// TIA Portal project "RollDice" (V17)

(* hardware
DEVICE "HMI_1"  TP1500 Comfort
   slot 0: "HMI_1"  TP1500 Comfort  6AV2 124-0QC02-0AX0  17.0.0.0
   slot 1: "HMI_RT_1"  TP1500 Comfort  6AV2 124-0QC02-0AX0  17.0.0.0
   slot 5: "HMI_1.IE_CP_1"  PROFINET Interface  17.0.0.0
      slot 1: "PROFINET Interface_1"  PROFINET Interface
         slot 1: "Port_1"  Port
         slot 2: "Port_2"  Port
   slot 6: "HMI_1.IE_CP_2"  PROFINET Interface  17.0.0.0
      slot 1: "PROFINET Interface_GBit"  PROFINET Interface
         slot 1: "Port_1"  Port
   slot 7: "HMI_1.MPI/DP_CP_1"  MPI/DP Interface  17.0.0.0
DEVICE "S7-1500/ET200MP station_1"  S7-1500 station
   slot 0: "Rail_0"  Rack  6ES7 590-1***0-0AA0
   slot 1: "PLC_1"  CPU 1515-2 PN  6ES7 515-2AM02-0AB0  V2.9
      slot 3: "CPU display_1"  6ES7591-1BA00-0AA0
      slot 32768: "PROFINET interface_1"  X1
         slot 32769: "Port_1"  X1 P1
         slot 32770: "Port_2"  X1 P2
      slot 33024: "PROFINET interface_2"  X2
         slot 33025: "Port_1"  X2 P1
      slot 34817: "Virtual CP interface port_1"  Virtual CP interface port  Virtual CP interface port
*)

// ===== PLC "PLC_1"  CPU 1515-2 PN =====

TYPE "Dice_PLCD"
   STRUCT
      Number : Int;   // 1-6 => Number on the Dice
      xRolled : Bool;   // True=> Dice has been clicked
   END_STRUCT;
END_TYPE

DATA_BLOCK "MainDB"   // DB1
{ S7_Optimized_Access := 'TRUE' }
VERSION : 0.1
   VAR
      Dice : Array[0..6] of "Dice_PLCD";
   END_VAR
BEGIN
END_DATA_BLOCK

FUNCTION "Dice_FC" : Void   // FC1, SCL
{ S7_Optimized_Access := 'TRUE' }
VERSION : 0.1
   VAR_OUTPUT
      error : Bool;   // Error if true
      status : Word;   // Status of the function
      subfunctionStatus : Word;   // Status or return value of called FB's, FCs and system blocks
   END_VAR
   VAR_IN_OUT
      Dice : "Dice_PLCD";
   END_VAR
   VAR_TEMP
      tempTime : DTL;   // System time
      tempNanoSecondInDWord : DWord;   // UDINT converted to DWORD for access to individual bytes
      tempTimeStatus : Word;   // Status of the instruction RD_SYS_T
      tempRandomValue : DWord;   // Random-start-value
      tempNormReal : Real;   // Normalized value
   END_VAR
   VAR CONSTANT
      ZERO : Int := 0;   // Zero value in case of error
      MAX_UDINT : UDInt := 4294967295 ;   // Maximum UDINT value
      SUB_STATUS_NO_ERROR : Word := 16#0000;   // Status: sub function call ends without error
      STATUS_FINISHED_NO_ERROR : Word := 16#0000;   // Status: Execution finished without errors
      ERR_MAX_LESS_MIN : Word := 16#8200;   // Error: The maximum limit number is smaller than the minimum limit number
      ERR_RD_SYS_T : Word := 16#8600;   // Error: System function Read system time returned an error
      LOWEST_NUMBER : UDInt := 1;   // Lowest Number a Dive can Roll
      HIGHEST_NUMBER : UDInt := 6;   // Highest Number a Dive can Roll
   END_VAR
BEGIN
   REGION Block_Header
       // Statement section REGION

   END_REGION

   REGION Validation

       // When not Rolled Jump Out of the Block
       IF #Dice.xRolled <> TRUE THEN
           RETURN;
       END_IF;


       // Read system time
       #tempTimeStatus := INT_TO_WORD(RD_SYS_T(#tempTime));

       // Check return variable for error
       IF (#tempTimeStatus <> #SUB_STATUS_NO_ERROR) THEN
           #error := true;
           #status := #ERR_RD_SYS_T;
           #subfunctionStatus := #tempTimeStatus;
           #Dice.Number := #ZERO;
           RETURN;
       END_IF;
   END_REGION

   REGION Calculating random number
       // Converting to double word so individual bytes can be addressed
       #tempNanoSecondInDWord := UDINT_TO_DWORD(#tempTime.NANOSECOND);

       // Callculate a random-start-value depending on the time
       #tempRandomValue.%B3 := #tempNanoSecondInDWord.%B0;
       #tempRandomValue.%B2 := #tempNanoSecondInDWord.%B1;
       #tempRandomValue.%B1 := #tempNanoSecondInDWord.%B2;
       #tempRandomValue.%B0 := #tempNanoSecondInDWord.%B3;
       // Norm the calculated random number: 0.0 <= #tempNormReal <= 1.0
       #tempNormReal := UDINT_TO_REAL(DWORD_TO_UDINT(#tempRandomValue)) / UDINT_TO_REAL(#MAX_UDINT);

       // Scale the tempNormReal to be in the range of maxValue and minValue
       #Dice.Number := REAL_TO_INT((#tempNormReal * UDINT_TO_REAL(#HIGHEST_NUMBER - #LOWEST_NUMBER) + UDINT_TO_REAL(#LOWEST_NUMBER)));
       #Dice.xRolled := FALSE;
       #error := false;
       #status := #STATUS_FINISHED_NO_ERROR;
       #subfunctionStatus := #SUB_STATUS_NO_ERROR;

       // ENO mechanism is not used
       ENO := TRUE;
   END_REGION
END_FUNCTION

ORGANIZATION_BLOCK "Main"   // OB1, FBD, ProgramCycle
TITLE = "Main Program Sweep (Cycle)"
{ S7_Optimized_Access := 'TRUE' }
VERSION : 0.1
   VAR_INPUT
      Initial_Call : Bool;   // Initial call of this OB
      Remanence : Bool;   // =True, if remanent data are available
   END_VAR
   VAR_TEMP
      Error : Word;
      xError : Bool;
   END_VAR
   VAR_TEMP   // added for the SCL form of the ladder/FBD networks
      _w1 : Bool;
      _w2 : Bool;
      _w3 : Bool;
      _w4 : Bool;
   END_VAR
BEGIN

REGION Network 1: True=> Dice has been clicked
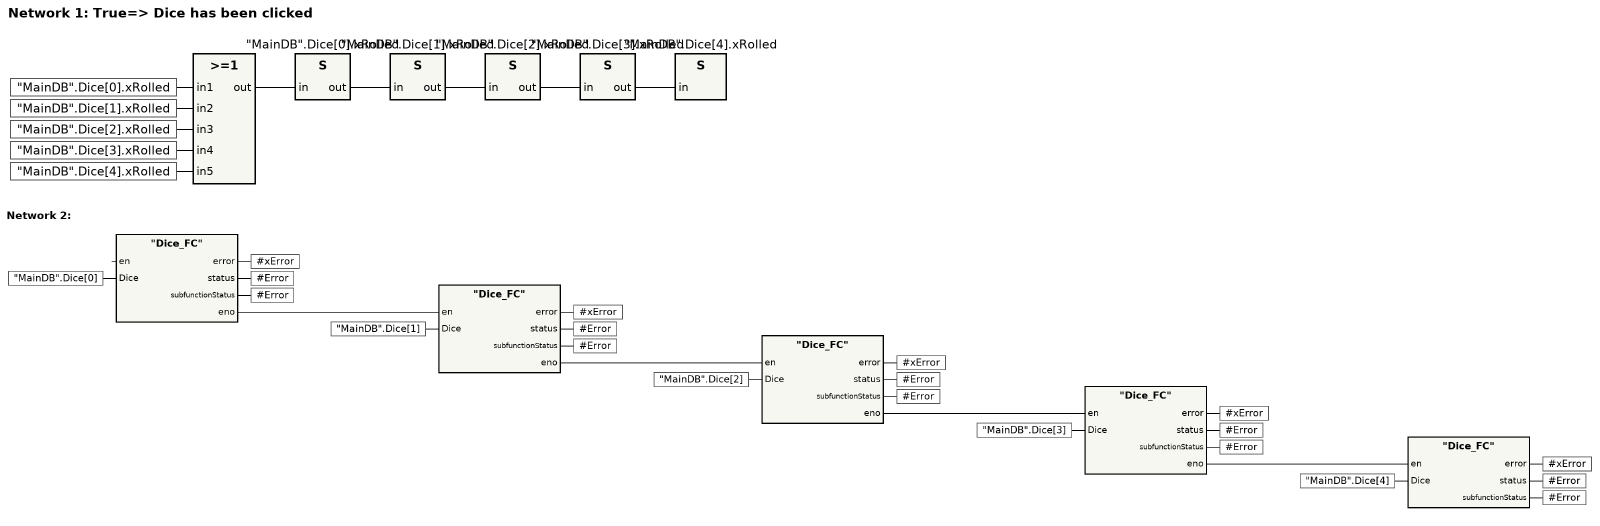
   #_w1 := "MainDB".Dice[0].xRolled OR "MainDB".Dice[1].xRolled OR "MainDB".Dice[2].xRolled OR "MainDB".Dice[3].xRolled OR "MainDB".Dice[4].xRolled;
   IF #_w1 THEN
       "MainDB".Dice[0].xRolled := TRUE;
       "MainDB".Dice[1].xRolled := TRUE;
       "MainDB".Dice[2].xRolled := TRUE;
       "MainDB".Dice[3].xRolled := TRUE;
       "MainDB".Dice[4].xRolled := TRUE;
   END_IF;
END_REGION

REGION Network 2
   "Dice_FC"(Dice := "MainDB".Dice[0],
             error => #xError,
             status => #Error,
             subfunctionStatus => #Error,
             ENO => #_w1);
   "Dice_FC"(EN := #_w1,
             Dice := "MainDB".Dice[1],
             error => #xError,
             status => #Error,
             subfunctionStatus => #Error,
             ENO => #_w2);
   "Dice_FC"(EN := #_w2,
             Dice := "MainDB".Dice[2],
             error => #xError,
             status => #Error,
             subfunctionStatus => #Error,
             ENO => #_w3);
   "Dice_FC"(EN := #_w3,
             Dice := "MainDB".Dice[3],
             error => #xError,
             status => #Error,
             subfunctionStatus => #Error,
             ENO => #_w4);
   IF #_w4 THEN
       "Dice_FC"(Dice := "MainDB".Dice[4], error => #xError, status => #Error, subfunctionStatus => #Error);
   END_IF;
END_REGION
END_ORGANIZATION_BLOCK

// ===== library types =====

// folder: LGF/4 Math operations

FUNCTION "LGF_RandomRange_Dint" : DInt   // FC10013, SCL
TITLE = LGF_RandomRange_DInt
{ S7_Optimized_Access := 'TRUE' }
AUTHOR : Siemens_Digital_Industries
FAMILY : LGF
NAME : LGF_RandomRange_DInt
// This function generates random numbers in defined limits (Datatype DInt)
   VAR_INPUT
      minValue : DInt;   // minimal Value random can reach / Minimum value of the range of the random number
      maxValue : DInt;   // maximal Value random can reach / Maximum value of the range of the random number
   END_VAR
   VAR_OUTPUT
      error : Bool;   // Error if true
      status : Word;   // Status of the function
      subfunctionStatus : Word;   // Status or return value of called FB's, FCs and system blocks
   END_VAR
   VAR_TEMP
      tempTime : DTL;   // System time
      tempNanoSecondInDWord : DWord;   // UDINT converted to DWORD for access to individual bytes
      tempTimeStatus : Word;   // Status of the instruction RD_SYS_T
      tempRandomValue : DWord;   // Random-start-value
      tempNormReal : Real;   // Normalized value
   END_VAR
   // Ret_Val : Returns random DInt number in a predefined range
   VAR CONSTANT
      ZERO : DInt := 0;   // Zero value in case of error
      MAX_UDINT : UDInt := 4294967295 ;   // Maximum UDINT value
      SUB_STATUS_NO_ERROR : Word := 16#0000;   // Status: sub function call ends without error
      STATUS_FINISHED_NO_ERROR : Word := 16#0000;   // Status: Execution finished without errors
      ERR_MAX_LESS_MIN : Word := 16#8200;   // Error: The maximum limit number is smaller than the minimum limit number
      ERR_RD_SYS_T : Word := 16#8600;   // Error: System function Read system time returned an error
   END_VAR
BEGIN
   REGION Block info header
     //=============================================================================
     // SIEMENS AG / (c)Copyright 2017
     //-----------------------------------------------------------------------------
     // Title:            LGF_RandomRange_DInt
     // Comment/Function: This function generates random numbers in defined limits (Datatype DInt)
     // Library/Family:   LGF(Library General Functions)
     // Author:           Siemens Digital Industry Support
     // Tested with:      S7-PLCSIM Advanced V2.0 SP1
     // Engineering:      TIA Portal V15 Update 2
     // Restrictions:     ENO disabled - error handling done by error and status
     // Requirements:     PLC (S7-1200 / S7-1500)
     //-------------------------------------------------------------------------------
     // Change log table:
     // Version  | Date       | Expert in charge       | Changes applied
     //----------|------------|------------------------|------------------------------
     // 01.00.00 19.08.2015  Siemens Industry Online Support
     //                      First released version
     // 01.00.01 02.01.2017  Siemens Industry Online Support
     //                      Upgrade: TIA Portal V14 Update 1
     // 01.00.02 17.08.2018  Siemens Industry Online Support
     //                      Upgrade: TIA V15 Update 2
     // 01.00.03 23.11.2018  Siemens Industry Online Support
     //                      Upgrade: TIA V15.1
     // 01.01.00 09.10.2019  Siemens Industry Presales Support
     //                      Renamed from "LGF_RandomInt" to "LGF_RandomRange_DInt"
     //                      change random datatype from int to dint
     //                      Regions, commens and costants are added
     // 03.00.00 23.04.2020  Siemens Industry Support
     //                      Set version to V3.0.0, harmonize the version of the whole library
     //=============================================================================
   END_REGION

   REGION Validation
     // Check if the maximal Value is less than the minimal value
     IF (#minValue > #maxValue) THEN
       #error := true;
       #status := #ERR_MAX_LESS_MIN;
       #subfunctionStatus := #SUB_STATUS_NO_ERROR;
       #LGF_RandomRange_DInt := #ZERO;
       RETURN;
     END_IF;

     // Read system time
     #tempTimeStatus := INT_TO_WORD(RD_SYS_T(#tempTime));

     // Check return variable for error
     IF (#tempTimeStatus <> #SUB_STATUS_NO_ERROR) THEN
       #error := true;
       #status := #ERR_RD_SYS_T;
       #subfunctionStatus := #tempTimeStatus;
       #LGF_RandomRange_DInt := #ZERO;
       RETURN;
     END_IF;
   END_REGION

   REGION Calculating random number
     // Converting to double word so individual bytes can be addressed
     #tempNanoSecondInDWord := UDINT_TO_DWORD(#tempTime.NANOSECOND);

     // Callculate a random-start-value depending on the time
     #tempRandomValue.%B3 := #tempNanoSecondInDWord.%B0;
     #tempRandomValue.%B2 := #tempNanoSecondInDWord.%B1;
     #tempRandomValue.%B1 := #tempNanoSecondInDWord.%B2;
     #tempRandomValue.%B0 := #tempNanoSecondInDWord.%B3;

     // Norm the calculated random number: 0.0 <= #tempNormReal <= 1.0
     #tempNormReal := UDINT_TO_REAL(DWORD_TO_UDINT(#tempRandomValue)) / UDINT_TO_REAL(#MAX_UDINT);

     // Scale the tempNormReal to be in the range of maxValue and minValue
     #LGF_RandomRange_DInt := REAL_TO_DINT((#tempNormReal * DINT_TO_REAL(#maxValue - #minValue) + DINT_TO_REAL(#minValue)));

     #error := false;
     #status := #STATUS_FINISHED_NO_ERROR;
     #subfunctionStatus := #SUB_STATUS_NO_ERROR;
     // ENO mechanism is not used
     ENO := TRUE;
   END_REGION
END_FUNCTION

FUNCTION "LGF_Random_UDInt" : UDInt   // FC10075, SCL
TITLE = LGF_Random_UDInt
{ S7_Optimized_Access := 'TRUE' }
AUTHOR : Siemens_Digital_Industries
FAMILY : LGF
NAME : LGF_Random_UDInt
// Generates a random number in the UDInt Range
   VAR_OUTPUT
      error : Bool;   // Error if true
      status : Word;   // Status of the function
      subfunctionStatus : Word;   // Status or return value of called FB's, FCs and system blocks
   END_VAR
   VAR_TEMP
      tempTime : DTL;   // System time
      tempNanoSecondInDWord : DWord;   // UDINT converted to DWORD for access to individual bytes
      tempTimeStatus : Word;   // Status of the instruction RD_SYS_T
      tempRandomValue : DWord;   // Random-start-value
   END_VAR
   // Ret_Val : Random number in the Dint range
   VAR CONSTANT
      ZERO : UDInt := 0;   // Zero value in case of error
      SUB_STATUS_NO_ERROR : Word := 16#0000;   // Status: No error / Initialize status
      STATUS_FINISHED_NO_ERROR : Word := 16#0000;   // Status: Execution finished without errors
      ERR_RD_SYS_T : Word := 16#8600;   // Error: System function Read system time returned an error
   END_VAR
BEGIN
   REGION Block info header
     //=============================================================================
     // SIEMENS AG / (c)Copyright 2019
     //-----------------------------------------------------------------------------
     // Title:            LGF_Random_UDInt
     // Comment/Function: Generates a random number in the UDInt Range
     // Library/Family:   LGF(Library General Functions)
     // Author:           Siemens Digital Industry Support
     // Tested with:      S7-PLCSIM Advanced V2.0 SP1
     // Engineering:      TIA Portal V15 Update 2
     // Restrictions:     ENO disabled - error handling done by error and status
     // Requirements:     PLC (S7-1200 / S7-1500)
     //-------------------------------------------------------------------------------
     // Change log table:
     // Version  | Date       | Expert in charge       | Changes applied
     //----------|------------|------------------------|------------------------------
     // 01.00.00 11.12.2019  Siemens Industry Presales Support
     //                      First release
     //                      copied from "LGF_Random_Real"
     // 03.00.00 23.04.2020  Siemens Industry Support
     //                      Set version to V3.0.0, harmonize the version of the whole library
     //=============================================================================
   END_REGION

   REGION Validation
     // Read system time
     #tempTimeStatus := INT_TO_WORD(RD_SYS_T(#tempTime));

     // Check return variable for error
     IF (#tempTimeStatus <> #SUB_STATUS_NO_ERROR) THEN
       #error := true;
       #status := #ERR_RD_SYS_T;
       #subfunctionStatus := #tempTimeStatus;
       #LGF_Random_UDInt := #ZERO;
       RETURN;
     END_IF;
   END_REGION

   REGION Calculating random number
     // Converting to double word so individual bytes can be addressed
     #tempNanoSecondInDWord := UDINT_TO_DWORD(#tempTime.NANOSECOND);

     // Calculate a random-start-value depending on the time
     #tempRandomValue.%B3 := #tempNanoSecondInDWord.%B0;
     #tempRandomValue.%B2 := #tempNanoSecondInDWord.%B1;
     #tempRandomValue.%B1 := #tempNanoSecondInDWord.%B2;
     #tempRandomValue.%B0 := #tempNanoSecondInDWord.%B3;

     #LGF_Random_UDInt := DWORD_TO_UDINT(#tempRandomValue);

     #error := false;
     #status := #STATUS_FINISHED_NO_ERROR;
     #subfunctionStatus := #SUB_STATUS_NO_ERROR;
     // ENO mechanism is not used
     ENO := TRUE;
   END_REGION
END_FUNCTION

(* ===== HMI "HMI_RT_1" =====
system functions are stored by id; their names below are inferred from use
connection "HMI_Connection_1": ETHERNET, S7_1500_OMS

HMI tags "Default tag table"
   "MainDB_Dice{0}" : Dice_PLCD = PLC MainDB.Dice[0], 100 ms
   "MainDB_Dice{1}" : Dice_PLCD = PLC MainDB.Dice[1], 100 ms
   "MainDB_Dice{2}" : Dice_PLCD = PLC MainDB.Dice[2], 100 ms
   "MainDB_Dice{3}" : Dice_PLCD = PLC MainDB.Dice[3], 100 ms
   "MainDB_Dice{4}" : Dice_PLCD = PLC MainDB.Dice[4], 100 ms

Template "Template_1" 1280x800
   Button "Exit" at 1200,739 size 78x59; TextOff 'Exit'; PictureOff "ExitRuntime_TP1500_Comfort_TR"; PictureOn "ExitRuntime_TP1500_Comfort_TR"
      on Release: StopRuntime(0)
   Button "Template_Button" at 1120,739 size 78x59; TextOff 'Text'
   Button "Template_Button_1" at 1040,739 size 78x59; TextOff 'Text'
   Button "Template_Button_2" at 960,739 size 78x59; TextOff 'Text'
   Button "Template_Button_3" at 880,739 size 78x59; TextOff 'Text'
   Button "Template_Button_4" at 800,739 size 78x59; TextOff 'Text'
   Button "Template_Button_5" at 720,739 size 78x59; TextOff 'Text'
   Button "Template_Button_6" at 640,739 size 78x59; TextOff 'Text'
   Button "Template_Button_7" at 561,739 size 78x59; TextOff 'Text'
   Button "Template_Button_8" at 481,739 size 78x59; TextOff 'Text'
   Button "Template_Button_9" at 401,739 size 78x59; TextOff 'Text'
   Button "Template_Button_10" at 321,739 size 78x59; TextOff 'Text'
   Button "Template_Button_11" at 241,739 size 78x59; TextOff 'Text'
   Button "Template_Button_12" at 161,739 size 78x59; TextOff 'Text'
   Button "Template_Button_13" at 81,739 size 78x59; TextOff 'Text'
   Button "Start screen" at 1,739 size 78x59; TextOff 'Start screen'; PictureOff "NavigateHome_TP1500_Comfort_TR"; PictureOn "NavigateHome_TP1500_Comfort_TR"
      on Release: ActivateScreen("Root screen", 0)

screen "Root screen" 1280x800, template "Template_1"
   TextField "HmiScreenItemData" at 128,354 size 1024x27; Text 'Welcome to HMI_1 (TP1500 Comfort)!'
   ScreenModuleView "Dice_1" at 186,142 size 150x150; ScreenModuleType ""
      Guid_{11997190-3445} <- "MainDB_Dice{0}"
   ScreenModuleView "Dice_2" at 350,142 size 150x150; ScreenModuleType ""
      Guid_{11997190-3445} <- "MainDB_Dice{1}"
   ScreenModuleView "Dice_3" at 514,142 size 150x150; ScreenModuleType ""
      Guid_{11997190-3445} <- "MainDB_Dice{2}"
   ScreenModuleView "Dice_4" at 678,142 size 150x150; ScreenModuleType ""
      Guid_{11997190-3445} <- "MainDB_Dice{3}"
   ScreenModuleView "Dice_5" at 842,142 size 150x150; ScreenModuleType ""
      Guid_{11997190-3445} <- "MainDB_Dice{4}"
*)

(* ===== HMI "HMI_RT_1" =====
system functions are stored by id; their names below are inferred from use

ScreenModuleEditorView "Dice" 640x480
   Circle "Number_1" at 65,65 size 40x40
      Visibility <- "Dice_PLCD.Number"
   Circle "Number_2_1" at 35,65 size 40x40
      Visibility <- "Dice_PLCD.Number"
   Circle "Number_2_2" at 95,65 size 40x40
      Visibility <- "Dice_PLCD.Number"
   Circle "Number_3_1" at 65,65 size 40x40
      Visibility <- "Dice_PLCD.Number"
   Circle "Number_3_2" at 35,100 size 40x40
      Visibility <- "Dice_PLCD.Number"
   Circle "Number_3_3" at 95,30 size 40x40
      Visibility <- "Dice_PLCD.Number"
   Circle "Number_4_1" at 35,90 size 40x40
      Visibility <- "Dice_PLCD.Number"
   Circle "Number_4_2" at 95,90 size 40x40
      Visibility <- "Dice_PLCD.Number"
   Circle "Number_4_3" at 35,40 size 40x40
      Visibility <- "Dice_PLCD.Number"
   Circle "Number_4_4" at 95,40 size 40x40
      Visibility <- "Dice_PLCD.Number"
   Circle "Number_5_1" at 30,95 size 40x40
      Visibility <- "Dice_PLCD.Number"
   Circle "Number_5_2" at 100,95 size 40x40
      Visibility <- "Dice_PLCD.Number"
   Circle "Number_5_3" at 30,35 size 40x40
      Visibility <- "Dice_PLCD.Number"
   Circle "Number_5_4" at 100,35 size 40x40
      Visibility <- "Dice_PLCD.Number"
   Circle "Number_5_5" at 65,65 size 40x40
      Visibility <- "Dice_PLCD.Number"
   Circle "Number_6_1" at 20,95 size 40x40
      Visibility <- "Dice_PLCD.Number"
   Circle "Number_6_2" at 110,95 size 40x40
      Visibility <- "Dice_PLCD.Number"
   Circle "Number_6_3" at 20,35 size 40x40
      Visibility <- "Dice_PLCD.Number"
   Circle "Number_6_4" at 110,35 size 40x40
      Visibility <- "Dice_PLCD.Number"
   Circle "Number_6_5" at 65,35 size 40x40
      Visibility <- "Dice_PLCD.Number"
   Circle "Number_6_6" at 65,95 size 40x40
      Visibility <- "Dice_PLCD.Number"
   Button "Button_1" at 10,10 size 150x150; TextOff 'Text'
      on Press: SetBit("Dice_PLCD.xRolled")
*)

(* ===== HMI "HMI_RT_1" =====
system functions are stored by id; their names below are inferred from use

ScreenModuleEditorView "Dice" 640x480
   Circle "Number_1" at 65,65 size 40x40
      Visibility <- "Dice_PLCD.Number"
   Circle "Number_2_1" at 35,65 size 40x40
      Visibility <- "Dice_PLCD.Number"
   Circle "Number_2_2" at 95,65 size 40x40
      Visibility <- "Dice_PLCD.Number"
   Circle "Number_3_1" at 65,65 size 40x40
      Visibility <- "Dice_PLCD.Number"
   Circle "Number_3_2" at 35,100 size 40x40
      Visibility <- "Dice_PLCD.Number"
   Circle "Number_3_3" at 95,30 size 40x40
      Visibility <- "Dice_PLCD.Number"
   Circle "Number_4_1" at 30,95 size 40x40
      Visibility <- "Dice_PLCD.Number"
   Circle "Number_4_2" at 100,95 size 40x40
      Visibility <- "Dice_PLCD.Number"
   Circle "Number_4_3" at 30,35 size 40x40
      Visibility <- "Dice_PLCD.Number"
   Circle "Number_4_4" at 100,35 size 40x40
      Visibility <- "Dice_PLCD.Number"
   Circle "Number_5_1" at 30,95 size 40x40
      Visibility <- "Dice_PLCD.Number"
   Circle "Number_5_2" at 100,95 size 40x40
      Visibility <- "Dice_PLCD.Number"
   Circle "Number_5_3" at 30,35 size 40x40
      Visibility <- "Dice_PLCD.Number"
   Circle "Number_5_4" at 100,35 size 40x40
      Visibility <- "Dice_PLCD.Number"
   Circle "Number_5_5" at 65,65 size 40x40
      Visibility <- "Dice_PLCD.Number"
   Circle "Number_6_1" at 20,95 size 40x40
      Visibility <- "Dice_PLCD.Number"
   Circle "Number_6_2" at 110,95 size 40x40
      Visibility <- "Dice_PLCD.Number"
   Circle "Number_6_3" at 20,35 size 40x40
      Visibility <- "Dice_PLCD.Number"
   Circle "Number_6_4" at 110,35 size 40x40
      Visibility <- "Dice_PLCD.Number"
   Circle "Number_6_5" at 65,35 size 40x40
      Visibility <- "Dice_PLCD.Number"
   Circle "Number_6_6" at 65,95 size 40x40
      Visibility <- "Dice_PLCD.Number"
   Button "Button_1" at 10,10 size 150x150; TextOff 'Text'
      on Press: SetBit("Dice_PLCD.xRolled")
*)